PROGRAM PRG_SL1L0_POWER
VAR // fix linking to rtd in the following order Bottom - South - TOP - NORTH
    {attribute 'pytmc' := '
        pv: SL1L0:POWER
        io: io
    '}
    {attribute 'TcLinkTo' := '.RTD_Bottom_1.iRaw := TIIB[SL1L0-EL3202-E8]^RTD Inputs Channel 1^Value;
                              .RTD_Bottom_1.bError := TIIB[SL1L0-EL3202-E8]^RTD Inputs Channel 1^Status^Error;
                              .RTD_Bottom_1.bUnderrange := TIIB[SL1L0-EL3202-E8]^RTD Inputs Channel 1^Status^Underrange;
                              .RTD_Bottom_1.bOverrange := TIIB[SL1L0-EL3202-E8]^RTD Inputs Channel 1^Status^Overrange;
                              .RTD_Bottom_2.iRaw := TIIB[SL1L0-EL3202-E8]^RTD Inputs Channel 2^Value;
                              .RTD_Bottom_2.bError := TIIB[SL1L0-EL3202-E8]^RTD Inputs Channel 2^Status^Error;
                              .RTD_Bottom_2.bUnderrange := TIIB[SL1L0-EL3202-E8]^RTD Inputs Channel 2^Status^Underrange;
                              .RTD_Bottom_2.bOverrange := TIIB[SL1L0-EL3202-E8]^RTD Inputs Channel 2^Status^Overrange;
                              .RTD_South_1.iRaw := TIIB[SL1L0-EL3202-E9]^RTD Inputs Channel 1^Value;
                              .RTD_South_1.bError := TIIB[SL1L0-EL3202-E9]^RTD Inputs Channel 1^Status^Error;
                              .RTD_South_1.bUnderrange := TIIB[SL1L0-EL3202-E9]^RTD Inputs Channel 1^Status^Underrange;
                              .RTD_South_1.bOverrange := TIIB[SL1L0-EL3202-E9]^RTD Inputs Channel 1^Status^Overrange;
                              .RTD_South_2.iRaw := TIIB[SL1L0-EL3202-E9]^RTD Inputs Channel 2^Value;
                              .RTD_South_2.bError := TIIB[SL1L0-EL3202-E9]^RTD Inputs Channel 2^Status^Error;
                              .RTD_South_2.bUnderrange := TIIB[SL1L0-EL3202-E9]^RTD Inputs Channel 2^Status^Underrange;
                              .RTD_South_2.bOverrange := TIIB[SL1L0-EL3202-E9]^RTD Inputs Channel 2^Status^Overrange;
                              .RTD_TOP_1.iRaw := TIIB[SL1L0-EL3202-E10]^RTD Inputs Channel 1^Value;
                              .RTD_TOP_1.bError := TIIB[SL1L0-EL3202-E10]^RTD Inputs Channel 1^Status^Error;
                              .RTD_TOP_1.bUnderrange := TIIB[SL1L0-EL3202-E10]^RTD Inputs Channel 1^Status^Underrange;
                              .RTD_TOP_1.bOverrange := TIIB[SL1L0-EL3202-E10]^RTD Inputs Channel 1^Status^Overrange;
                              .RTD_TOP_2.iRaw := TIIB[SL1L0-EL3202-E10]^RTD Inputs Channel 2^Value;
                              .RTD_TOP_2.bError := TIIB[SL1L0-EL3202-E10]^RTD Inputs Channel 2^Status^Error;
                              .RTD_TOP_2.bUnderrange := TIIB[SL1L0-EL3202-E10]^RTD Inputs Channel 2^Status^Underrange;
                              .RTD_TOP_2.bOverrange := TIIB[SL1L0-EL3202-E10]^RTD Inputs Channel 2^Status^Overrange;
                              .RTD_North_1.iRaw := TIIB[SL1L0-EL3202-E11]^RTD Inputs Channel 1^Value;
                              .RTD_North_1.bError := TIIB[SL1L0-EL3202-E11]^RTD Inputs Channel 1^Status^Error;
                              .RTD_North_1.bUnderrange := TIIB[SL1L0-EL3202-E11]^RTD Inputs Channel 1^Status^Underrange;
                              .RTD_North_1.bOverrange := TIIB[SL1L0-EL3202-E11]^RTD Inputs Channel 1^Status^Overrange;
                              .RTD_North_2.iRaw := TIIB[SL1L0-EL3202-E11]^RTD Inputs Channel 2^Value;
                              .RTD_North_2.bError := TIIB[SL1L0-EL3202-E11]^RTD Inputs Channel 2^Status^Error;
                              .RTD_North_2.bUnderrange := TIIB[SL1L0-EL3202-E11]^RTD Inputs Channel 2^Status^Underrange;
                              .RTD_North_2.bOverrange := TIIB[SL1L0-EL3202-E11]^RTD Inputs Channel 2^Status^Overrange'}
    fbSL1L0: FB_SLITS_POWER;

    {attribute 'pytmc' := '
    pv: SL1L0:POWER:GO;
    io: io;
    field: ZNAM False;
    field: ONAM True;
    '}
    bExecuteMotion:BOOL ;

    // Default True until it is properly linked to PMPS bit
    bMoveOk:BOOL :=TRUE;


    mcPower : ARRAY [1..4] OF MC_POWER;

        (*Offsets*)
    (* Absolute encoder value at the HLS + Absolute encoder value at the centered beam *)
    rEncoderOffsetTop: REAL := 15.55;
    rEncoderOffsetBottom: REAL := -12.99;
    rEncoderOffsetNorth: REAL := 12.2;
    rEncoderOffsetSouth: REAL := -16.8;

END_VAR



(*
--MAPPING TO PHYSICAL TERMINAL--
Main.41 -> M1    (Bottom)
Main.42 -> M2    (South)
Main.43 -> M3    (Top)
Main.44 -> M4    (North)
*)

fbSL1L0.rEncoderOffsetTop := rEncoderOffsetTop;
fbSL1L0.rEncoderOffsetBottom := rEncoderOffsetBottom;
fbSL1L0.rEncoderOffsetNorth := rEncoderOffsetNorth;
fbSL1L0.rEncoderOffsetSouth := rEncoderOffsetSouth;

//fbSL1L0.bExecuteMotion := bExecuteMotion;
fbSL1L0.bMoveOk := bMoveOk;
fbSL1L0(stTopBlade:=  Main.M43,
        stBottomBlade:= Main.M41,
        stNorthBlade:=  Main.M44,
        stSouthBlade:=  Main.M42,
        bExecuteMotion:=bExecuteMotion);

//for testing purposes only. comment-out/delete once done.
(*mcPower[1](axis:=Main.M41.Axis, Enable:=TRUE, enable_positive:=Main.M41.bLimitForwardEnable, enable_negative:=Main.M41.bLimitBackwardEnable);
mcPower[2](axis:=Main.M42.Axis, Enable:=TRUE, enable_positive:=Main.M42.bLimitForwardEnable, enable_negative:=Main.M42.bLimitBackwardEnable);
mcPower[3](axis:=Main.M43.Axis, Enable:=TRUE, enable_positive:=Main.M43.bLimitForwardEnable, enable_negative:=Main.M43.bLimitBackwardEnable);
mcPower[4](axis:=Main.M44.Axis, Enable:=TRUE, enable_positive:=Main.M44.bLimitForwardEnable, enable_negative:=Main.M44.bLimitBackwardEnable);*)

END_PROGRAM

(* stored: Version 1.1.0.1, ProductVersion 3.1.4022.18
   POU PRG_SL1L0_POWER: Id {bb2d6beb-8e46-4873-9e1c-8b32c60eb928}, SpecialFunc None *)
